INTERFACE PUBLIC IdleCommands

METHOD PUBLIC Abort
END_METHOD

METHOD PUBLIC Start
END_METHOD

METHOD PUBLIC Stop
END_METHOD

END_INTERFACE

(* stored: Version 1.1.0.1, ProductVersion 3.1.4026.12
   Itf IdleCommands: Id {98a18d41-1301-03fd-1f24-fccf520ed562}
   Method Abort: Id {0c7667c6-a706-494a-9950-a42bd0f9f67e}
   Method Start: Id {10ff5ee6-413f-0d0d-317f-29627efddc1f}
   Method Stop: Id {9afaa9a1-e547-484d-a795-ed679c222660} *)
